FUNCTION ProcessInitialization : E_PROGRESS
VAR_INPUT
  eVariant    : E_APP_VARIANT;
END_VAR
VAR
END_VAR


CASE eVariant
OF
  E_APP_VARIANT.VARIANT_OUTPUT_24:
    Initialization_Robot();
    ProcessInitialization                 := E_PROGRESS.PROGRESS_DONE;

  E_APP_VARIANT.VARIANT_OUTPUT_CLAMP:
    Initialization_Clamp();
    ProcessInitialization                 := E_PROGRESS.PROGRESS_DONE;

ELSE
    ProcessInitialization                 := E_PROGRESS.PROGRESS_INIT;
END_CASE

END_FUNCTION

(* stored: Version 1.1.0.1, ProductVersion 3.1.4026.13
   POU ProcessInitialization: Id {8ae0d3f5-bf9f-423d-bf28-ae364d3e015c}, SpecialFunc None *)
